// ---- FBs/FB_ECS_Keba_P30_noWrite.TcPOU
FUNCTION_BLOCK FB_ECS_Keba_P30_noWrite
VAR_INPUT PERSISTENT
	///{#lynus.ag#()} //Enable the Fuctionblock and his logic
	bEnable: BOOL;
	bEnable_write: BOOL;
	///With True its possible to invert all received power data from the electric meter
	bPowerDataInvers: BOOL;
	///Electric Fuse Line on wich the ECS is connected => 1 2 3 (If 0 then this charging station is not connected to a Electric Fuse Line)
	byElectricFuseLine: BYTE;
	///Failsafe Current when the connection between PLC and Charging station is interrupted. 0mA = CS Off, 6000mA - 32000mA
	uiFailsafeCurrent: UINT;
	///Failsafe Timeout when the connection between PLC and Charging station is interrupted. 10 - 600 sec
	uiFailsafeTimeOut: UINT := 10;
	///Number of EMS what control this Device.
	diNrOfEMS_IN: DINT;
	///Number of the electric meter for incoming power data. (Power Data for this Device)
	diNrOfEM_IN_CS: DINT;
	///IP Adress from the Keba charging station
	sIPAdress: STRING(15);
	///{#lynus.ag#()} //Setup charging station
	stSetupECS: ST_Setup_ECS;
END_VAR
VAR_OUTPUT
	///{#lynus.ag#()} //Electric charging station output data
	stDataECS: ST_ECS_Output;
	///Active Number from the Electric charging Function for using on other functions
	diNrOfECS_OUT: DINT;
	///Total Electric Power in kW read out directly from the Charging station. (Real time)
	lrTotalPowerECSRealTime: LREAL;
END_VAR
VAR
	///Function block for electric charging station

	fbCS: FB_ElectricChargingStation;
	///Function block to calcualte the number of the Device

	fbNumberDevice: FB_NumberOfDevice;
	///Digital Input from external loock signal
	fbDIExternalLock: FB_XL1XXX_DI;
	///Modbus Read Function (FC3)

	fbMBRead_FC3: FB_MBReadRegs;
	///Modbus Write Function (FC6)

	fbMBWrite_FC6: FB_MBWriteSingleReg;
	///Convert Word to Dword

	fbConvertWordToDword: FB_CV_WORD_TO_DWORD;
	///Timer for Delay between Requests

	timDelay: TON;
	///Timer for Timeout

	timTimeout: TON;
	///Timer to dissable the Function after Lynus_Standards.Constants_General.tTimeDissableLynusFunctions Days without connection to the Lynus Cloud

	timDissableFunctions: TON;
	///Timer to try reset the connection Flag on the GVL. (When somebody delete the Connection Function and make only a onlinechange)

	timResetConnectionOnGVL: TON;
	///Charging Time

	timChTimeSocket: TON;
	///Timer to start the state machine with Daley after enabling or after the system ist restartet

	timDelayStart: TON;
	///Timer to Close the Socket after to much Errors

	timCloseSocket: TON;
	///Internal positive Edge

	FPError_FC_3: R_TRIG;
	///Internal positive Edge

	FPError_FC_6: R_TRIG;
	///Internal positive Edge

	FPEnable: R_TRIG;
	///Function to save persistent data

	arrPD: ARRAY[1..16] OF FB_PersistentData_Number;
	///Function to save persistent string data

	fbPDString: FB_PersistentData_String;
	///Buffer with Data from FC3

	arrBuffer_FC3: ARRAY[1..2] OF WORD;
	///Error State from the charging station

	bErrorCS: BOOL;
	///Modbus TCP Function Error Counter																	

	byMBTCPErrorCounter: BYTE;
	///Wait in Step before start to clean data on PLC

	byWaitInStep: BYTE;
	///State machine to handle the data on the GVL

	iStateGVLData: INT;
	///State machine for read out Data over Modbus TCP

	iStateModbusRead: INT;
	///State machine for write Data over Modbus TCP

	iStateModbusWrite: INT;
	///State machine for error out Data over Modbus TCP	

	iStateModbusError: INT;
	///Variable to compare the state machine variable to set or reset the timeout timer

	iStateModbus_CP: INT;
	///Number of active batterys

	diNumberOfActiveBatterys: DINT;
	///Number of battery inverters that work in Emergency Power operation 

	diNumberOfBatteryInverterInEPO: DINT;
	///Loop to clean old data on GVL

	diLPForGVL: DINT;
	///Counter to clean old data on GVL

	diCounterForGVL: DINT;
	///Sum of the SOC from all batterys

	dwSumSOC: DWORD;
	///Charging State from the Keba Charger

	dwChargingState: DWORD;
	///Cable State from the Keba Charger

	dwCableState: DWORD;
	///Error Code from the Keba Charger

	dwErrorCode: DWORD;
	///Power from the ECS in W 

	rPowerECS: REAL;
	///Energy Counter Consumption in Wh

	lrTotalCounterEnergy_Consumption: LREAL;
	///Charged Energy from the active Session in Wh

	lrChargedEnergySession: LREAL;
	///Loop to check some data from batterys

	liLPBatteryData: LINT;
	///Loop to check if 1 or more battery inverters build a island grid

	liLPInEPO: LINT;
END_VAR
VAR PERSISTENT
	///Number of EMS what control this Device to compare with the original
	{attribute 'conditionalshow' := ''}
	diNrOfEMS_IN_CP: DINT;
END_VAR

//Creator : Stefan Lackner
//Company : EfficientIO
//Date : 14.05.2024
//Version : 1.0.0.1 based on V1.0.0.0

//With this Funcition its possible to communicate with a Keba P30 Charging station over Modbus TCP.
//Support the C-Series from Version 3.10.16 or higher
//Support the X-Series from Version 1.11 or higher
//Its possible to controll the charging station over the charge current
//When the Function send 0 Ampere is switched of, then the charging station is blocked and its not possible to charge
//The Communication is not so fast because in the Documentation they write that we can read every 500MS but we can write onle ever 5 seconds.
//We can read only 1 Register at each command. Its not possible to read more Registers with 1 command
//The Unit ID is always 255
//Also the Settings for Fail Save is includes in ths Fuction. The Failsave Current is set to uiFailsafeCurrent.
//Failsafe takes effect when the connection between the PLC and the charging station is interrupted. Timout is uiFailsafeTimeOut in seconds.

//Versions that are supported : 1.3

//NOTE for diNr.....Designation => 
//_IN = Here Data come in from other Functions or go out to other functions about the GVL
//_OUT = Here Data go out to other functions about the GVL

(*--------------------------------------------------------------------------------------------Limits-------------------------------------------------------------------------------------*)

diNrOfEMS_IN := LIMIT(0,diNrOfEMS_IN,Constants_Energy.diMaxNumberOfEMS);
diNrOfEM_IN_CS := LIMIT(0,diNrOfEM_IN_CS,Constants_Energy.diMaxNumberOfElectricMeters);
byElectricFuseLine := LIMIT(0,byElectricFuseLine,30);
IF uiFailsafeCurrent > 0 THEN 
	uiFailsafeCurrent := LIMIT(6000,uiFailsafeCurrent,32000);
END_IF 
uiFailsafeTimeOut := LIMIT(10,uiFailsafeTimeOut,600);	
		
(*------------------------------------------------------------------Power Data----------------------------------------------------------------------------*)

IF diNrOfEM_IN_CS <> 0 THEN
	//Energy Session Input data
	fbCS.bCalculateEnergySession := FALSE;
	fbCS.arrSocketPowerECS[1] := 0;
	fbCS.arrSocketPowerECS[2] := 0;
	fbCS.arrSocketPowerECS[3] := 0;
	fbCS.arrSocketPowerECS[4] := 0;
	fbCS.arrSocketEnergySession[1] := 0;
	fbCS.arrSocketEnergySession[2] := 0;
	fbCS.arrSocketEnergySession[3] := 0;
	fbCS.arrSocketEnergySession[4] := 0;
	IF NOT bPowerDataInvers THEN
		//Energy meter input data for cs Function block
		fbCS.lrCounterEnergyT1_Consumption := Lynus_Standards.GVL_Energy.stDataElectricMeters[diNrOfEM_IN_CS].lrCounterEnergyT1_Production * 1000;
		fbCS.lrCounterEnergyT2_Consumption := Lynus_Standards.GVL_Energy.stDataElectricMeters[diNrOfEM_IN_CS].lrCounterEnergyT2_Production * 1000;
		fbCS.lrCounterEnergyT1_Production := Lynus_Standards.GVL_Energy.stDataElectricMeters[diNrOfEM_IN_CS].lrCounterEnergyT1_Consumption * 1000;
		fbCS.lrCounterEnergyT2_Production := Lynus_Standards.GVL_Energy.stDataElectricMeters[diNrOfEM_IN_CS].lrCounterEnergyT1_Consumption * 1000;
		fbCS.lrTotalCounterEnergy_Consumption := Lynus_Standards.GVL_Energy.stDataElectricMeters[diNrOfEM_IN_CS].lrTotalCounterEnergy_Production * 1000;
		fbCS.lrTotalCounterEnergy_Production := Lynus_Standards.GVL_Energy.stDataElectricMeters[diNrOfEM_IN_CS].lrTotalCounterEnergy_Consumption * 1000;
		fbCS.lrTotalPowerECS := (Lynus_Standards.GVL_Energy.stDataElectricMeters[diNrOfEM_IN_CS].lrPower * 1000) * - 1;
	ELSE
		//Energy meter input data for cs Function block
		fbCS.lrCounterEnergyT1_Consumption := Lynus_Standards.GVL_Energy.stDataElectricMeters[diNrOfEM_IN_CS].lrCounterEnergyT1_Consumption * 1000;
		fbCS.lrCounterEnergyT2_Consumption := Lynus_Standards.GVL_Energy.stDataElectricMeters[diNrOfEM_IN_CS].lrCounterEnergyT2_Consumption * 1000;
		fbCS.lrCounterEnergyT1_Production := Lynus_Standards.GVL_Energy.stDataElectricMeters[diNrOfEM_IN_CS].lrCounterEnergyT1_Production * 1000;
		fbCS.lrCounterEnergyT2_Production := Lynus_Standards.GVL_Energy.stDataElectricMeters[diNrOfEM_IN_CS].lrCounterEnergyT2_Production * 1000;
		fbCS.lrTotalCounterEnergy_Consumption := Lynus_Standards.GVL_Energy.stDataElectricMeters[diNrOfEM_IN_CS].lrTotalCounterEnergy_Consumption * 1000;
		fbCS.lrTotalCounterEnergy_Production := Lynus_Standards.GVL_Energy.stDataElectricMeters[diNrOfEM_IN_CS].lrTotalCounterEnergy_Production * 1000;
		fbCS.lrTotalPowerECS := Lynus_Standards.GVL_Energy.stDataElectricMeters[diNrOfEM_IN_CS].lrPower * 1000;
	END_IF
ELSE
	//Energy meter input data for cs Function block
	fbCS.lrCounterEnergyT1_Consumption := lrTotalCounterEnergy_Consumption;
	fbCS.lrCounterEnergyT2_Consumption := 0;
	fbCS.lrCounterEnergyT1_Production := 0;
	fbCS.lrCounterEnergyT2_Production := 0;
	fbCS.lrTotalCounterEnergy_Consumption := lrTotalCounterEnergy_Consumption;
	fbCS.lrTotalCounterEnergy_Production := 0;
	fbCS.lrTotalPowerECS := rPowerECS;
	//Energy Session Input data
	fbCS.bCalculateEnergySession := FALSE;
	fbCS.arrSocketPowerECS[1] := rPowerECS;
	fbCS.arrSocketPowerECS[2] := 0;
	fbCS.arrSocketPowerECS[3] := 0;
	fbCS.arrSocketPowerECS[4] := 0;
	fbCS.arrSocketEnergySession[1] := lrChargedEnergySession;
	fbCS.arrSocketEnergySession[2] := 0;
	fbCS.arrSocketEnergySession[3] := 0;
	fbCS.arrSocketEnergySession[4] := 0;
END_IF			

(*-------------------------------------------------------------Calcualte the number of ECS---------------------------------------------------------------*)

fbNumberDevice(
	diActualNumberOfDevices:= Lynus_Standards.GVL_Energy.stNumberOfDevices.diNumberOfECS, 
	diMaxNumberOfDevices:= Constants_Energy.diMaxNumberOfElectricChargingStations, 
	udiCounterOnlineChange:= TwinCAT_SystemInfoVarList._AppInfo.OnlineChangeCnt, 
	bNumberIsCalculatet=> , 
	bFPNumberIsCalculatet=> , 
	bOnlineChange=> , 
	diNumberForThisDevice=> diNrOfECS_OUT, 
	diNumberOfTotalDevices=> );

//Write new Numer on GVL
IF fbNumberDevice.bFPNumberIsCalculatet THEN
	Lynus_Standards.GVL_Energy.stNumberOfDevices.diNumberOfECS := fbNumberDevice.diNumberOfTotalDevices;	
END_IF 

//Delete old Number on GVL
IF fbNumberDevice.bOnlineChange THEN 
	Lynus_Standards.GVL_Energy.stNumberOfDevices.diNumberOfECS := diNrOfECS_OUT;	
	iStateGVLData := 1;
END_IF

(*-------------------------------------------------------------Service from Backend is ready and check the connection to backen for dissabel/enable Function---------------------------------------------------------------*)

//Try to reset the variable for connection on the GVL. When all is normal then the Lynus Mqtt connection function set this variable to true in the next cycle
//When we have no connection to the backend then after Lynus_Standards.Constants_General.tTimeDissableLynusFunctions days the Function is dissabled with all of his functionalities
timResetConnectionOnGVL(IN:= NOT timResetConnectionOnGVL.Q, PT:= T#1H, Q=> , ET=> );
IF timResetConnectionOnGVL.Q THEN 
	Lynus_Standards.GVL_Communicator.bStateConnectionToEnableFunctions := FALSE; 
END_IF
IF NOT Lynus_Standards.GVL_Communicator.bStateConnectionToEnableFunctions THEN 
	timDissableFunctions.IN := TRUE; 
ELSE 
	timDissableFunctions.IN := FALSE; 
END_IF  
timDissableFunctions(	IN:= , 	
						PT:= Lynus_Standards.Constants_General.tTimeDissableLynusFunctions, 
						Q=> , 
						ET=> );
			
(*--------------------------------------------------------------------------------------------State Machine Read--------------------------------------------------------------------------------------*)

//Timer for Delay
timDelay(	IN:= , 
			PT:= T#750MS, 
			Q=> , 
			ET=> );

//Timer for Timeout in Statemachine
IF 	(iStateModbusRead > 0 AND iStateModbusRead <= 7 AND iStateModbusRead = iStateModbus_CP) OR
	(iStateModbusWrite > 0 AND iStateModbusWrite <= 2 AND iStateModbusWrite = iStateModbus_CP) THEN
		timTimeout.IN := TRUE;
ELSE	
		timTimeout.IN := FALSE;
END_IF
//Timeout Timer is dissabled when the Init Step is aktiv or the function is not enabled
IF (iStateModbusRead = 0 AND iStateModbusWrite = 0) OR NOT bEnable THEN 
	timTimeout.IN := FALSE; 
END_IF
timTimeout(	IN:= , 
			PT:= T#10S, 
			Q=> , 
			ET=> );

//Enable with Delay that not all sockets have to be created at the same time
timDelayStart(	IN:= bEnable, 
				PT:= T#20MS * diNrOfECS_OUT, 
				Q=> , 
				ET=> );
FPEnable(	CLK:= timDelayStart.Q, 
			Q=> );

IF FPEnable.Q AND iStateModbusRead = 0 AND iStateModbusWrite = 0 THEN 
	iStateModbusRead := 1; 
END_IF		
		
//Not Enabled
IF NOT bEnable THEN 
	iStateModbusRead := 0; 
	iStateModbusError := 0; 
	iStateModbusWrite := 0; 
END_IF		
		
CASE iStateModbusRead OF

	0://Init Step 
		iStateModbus_CP := 0;
		timDelay.IN := FALSE;
		fbMBRead_FC3.bExecute := FALSE;
		fbMBWrite_FC6.bExecute := FALSE;
		rPowerECS := 0;
		dwChargingState := 0;
		dwCableState := 0;	
		lrChargedEnergySession := 0;
	
	1://Charging State (Register 1000) !!!!Maybe 0 or 1....test it. Then change also the other Register Adresses!!!!!
		iStateModbus_CP := iStateModbusRead;

		//Start Read
		fbMBRead_FC3.nQuantity := 2;
		fbMBRead_FC3.nMBAddr := 1000;
		fbMBRead_FC3.bExecute := TRUE;
		fbMBRead_FC3.nUnitID := 255;
			
		IF fbMBRead_FC3.bBusy THEN 
			timDelay.IN := TRUE; 
		END_IF
		
		//Wait for Delay, copy Data and then next step
		IF NOT fbMBRead_FC3.bBusy AND NOT fbMBRead_FC3.bError AND timDelay.Q THEN
			//Charging State
			fbConvertWordToDword(wInputValue_1:= arrBuffer_FC3[1], wInputValue_2:= arrBuffer_FC3[2], eByteOrderForConvert:= eByteOrder.eBigEndian, dwOutputValue =>);
			dwChargingState := fbConvertWordToDword.dwOutputValue;
			
			//Go to Next Step
			fbMBRead_FC3.bExecute := FALSE;
			timDelay.IN := FALSE;		
			iStateModbusRead := 2;
		END_IF	

		//Error or Timeout
		IF FPError_FC_3.Q OR timTimeout.Q THEN
			iStateModbusError := 300;
		END_IF	
		
	2://Cable State (Register 1004)
		iStateModbus_CP := iStateModbusRead;

		//Start Read
		fbMBRead_FC3.nQuantity := 2;
		fbMBRead_FC3.nMBAddr := 1004;
		fbMBRead_FC3.bExecute := TRUE;
		fbMBRead_FC3.nUnitID := 255;
			
		IF fbMBRead_FC3.bBusy THEN 
			timDelay.IN := TRUE; 
		END_IF
		
		//Wait for Delay, copy Data and then next step
		IF NOT fbMBRead_FC3.bBusy AND NOT fbMBRead_FC3.bError AND timDelay.Q THEN
			//Cable State
			fbConvertWordToDword(wInputValue_1:= arrBuffer_FC3[1], wInputValue_2:= arrBuffer_FC3[2], eByteOrderForConvert:= eByteOrder.eBigEndian, dwOutputValue =>);
			dwCableState := fbConvertWordToDword.dwOutputValue;
			//Go to Next Step
			fbMBRead_FC3.bExecute := FALSE;
			timDelay.IN := FALSE;		
			iStateModbusRead := 3;
		END_IF	

		//Error or Timeout
		IF FPError_FC_3.Q OR timTimeout.Q THEN
			iStateModbusError := 300;
		END_IF	
		
	3://Error Code (Register 1006)
		iStateModbus_CP := iStateModbusRead;

		//Start Read
		fbMBRead_FC3.nQuantity := 2;
		fbMBRead_FC3.nMBAddr := 1006;
		fbMBRead_FC3.bExecute := TRUE;
		fbMBRead_FC3.nUnitID := 255;
			
		IF fbMBRead_FC3.bBusy THEN 
			timDelay.IN := TRUE; 
		END_IF
		
		//Wait for Delay, copy Data and then next step
		IF NOT fbMBRead_FC3.bBusy AND NOT fbMBRead_FC3.bError AND timDelay.Q THEN
			//Error Code
			fbConvertWordToDword(wInputValue_1:= arrBuffer_FC3[1], wInputValue_2:= arrBuffer_FC3[2], eByteOrderForConvert:= eByteOrder.eBigEndian, dwOutputValue =>);
			dwErrorCode := fbConvertWordToDword.dwOutputValue;
			//Go to Next Step
			fbMBRead_FC3.bExecute := FALSE;
			timDelay.IN := FALSE;		
			iStateModbusRead := 4;
		END_IF	

		//Error or Timeout
		IF FPError_FC_3.Q OR timTimeout.Q THEN
			iStateModbusError := 300;
		END_IF	
		
	4://Active Power (Register 1020)
		iStateModbus_CP := iStateModbusRead;

		//Start Read
		fbMBRead_FC3.nQuantity := 2;
		fbMBRead_FC3.nMBAddr := 1020;
		fbMBRead_FC3.bExecute := TRUE;
		fbMBRead_FC3.nUnitID := 255;
			
		IF fbMBRead_FC3.bBusy THEN 
			timDelay.IN := TRUE; 
		END_IF
		
		//Wait for Delay, copy Data and then next step
		IF NOT fbMBRead_FC3.bBusy AND NOT fbMBRead_FC3.bError AND timDelay.Q THEN
			//Active Power in mW
			fbConvertWordToDword(wInputValue_1:= arrBuffer_FC3[1], wInputValue_2:= arrBuffer_FC3[2], eByteOrderForConvert:= eByteOrder.eBigEndian, dwOutputValue =>);
			rPowerECS := DWORD_TO_REAL(fbConvertWordToDword.dwOutputValue);
			rPowerECS := rPowerECS / 1000;	
			//Go to Next Step
			fbMBRead_FC3.bExecute := FALSE;
			timDelay.IN := FALSE;		
			iStateModbusRead := 5;
		END_IF	

		//Error or Timeout
		IF FPError_FC_3.Q OR timTimeout.Q THEN
			iStateModbusError := 300;
		END_IF	
	
	5://Total Energy (Register 1036)
		iStateModbus_CP := iStateModbusRead;

		//Start Read
		fbMBRead_FC3.nQuantity := 2;
		fbMBRead_FC3.nMBAddr := 1036;
		fbMBRead_FC3.bExecute := TRUE;
		fbMBRead_FC3.nUnitID := 255;
			
		IF fbMBRead_FC3.bBusy THEN 
			timDelay.IN := TRUE; 
		END_IF
		
		//Wait for Delay, copy Data and then next step
		IF NOT fbMBRead_FC3.bBusy AND NOT fbMBRead_FC3.bError AND timDelay.Q THEN
			//Total Energy in Wh
			fbConvertWordToDword(wInputValue_1:= arrBuffer_FC3[1], wInputValue_2:= arrBuffer_FC3[2], eByteOrderForConvert:= eByteOrder.eBigEndian, dwOutputValue =>);
			lrTotalCounterEnergy_Consumption := DWORD_TO_LREAL(fbConvertWordToDword.dwOutputValue);
			//Go to Next Step
			fbMBRead_FC3.bExecute := FALSE;
			timDelay.IN := FALSE;		
			iStateModbusRead := 6;
		END_IF	

		//Error or Timeout
		IF FPError_FC_3.Q OR timTimeout.Q THEN
			iStateModbusError := 300;
		END_IF	
		
	6://Charged Energy from current charging session (Register 1502)
		iStateModbus_CP := iStateModbusRead;

		//Start Read
		fbMBRead_FC3.nQuantity := 2;
		fbMBRead_FC3.nMBAddr := 1502;
		fbMBRead_FC3.bExecute := TRUE;
		fbMBRead_FC3.nUnitID := 255;
			
		IF fbMBRead_FC3.bBusy THEN 
			timDelay.IN := TRUE; 
		END_IF
		
		//Wait for Delay, copy Data and then next step
		IF NOT fbMBRead_FC3.bBusy AND NOT fbMBRead_FC3.bError AND timDelay.Q THEN
			//Total Energy in Wh
			fbConvertWordToDword(wInputValue_1:= arrBuffer_FC3[1], wInputValue_2:= arrBuffer_FC3[2], eByteOrderForConvert:= eByteOrder.eBigEndian, dwOutputValue =>);
			lrChargedEnergySession := DWORD_TO_LREAL(fbConvertWordToDword.dwOutputValue);
			//Go to Next Step
			fbMBRead_FC3.bExecute := FALSE;
			timDelay.IN := FALSE;		
			iStateModbusRead := 7;
		END_IF	

		//Error or Timeout
		IF FPError_FC_3.Q OR timTimeout.Q THEN
			iStateModbusError := 300;
		END_IF	
		
	7://Wait 1 Step to reset the delay counter befor start to write
		iStateModbus_CP := iStateModbusRead;
		IF bEnable_write THEN 
			iStateModbusWrite := 1;
			//-1 because 0 is the Init Step for Read
			iStateModbusRead := - 1;
		ELSE
			iStateModbusRead := 1;
		END_IF				
		//Error on Master, changes on Inputs or Timeout
		IF timTimeout.Q THEN 
			iStateModbusError := 300;	 
		END_IF

END_CASE

(*------------------------------------------------------------------Error and Warning----------------------------------------------------------------------------*)	
 
IF dwChargingState = 4 OR dwErrorCode <> 0 THEN 
	bErrorCS := TRUE; 
ELSE 
	bErrorCS := FALSE; 
END_IF

IF timDissableFunctions.Q THEN 
	fbCS.bWarning := TRUE; 
	fbCS.iWarningCode := 0; 
ELSE 
	fbCS.bWarning := FALSE; 
END_IF   
IF Lynus_Standards.GVL_Energy.stNumberOfDevices.diNumberOfECS > Constants_Energy.diMaxNumberOfElectricChargingStations OR bErrorCS OR byMBTCPErrorCounter > 10 THEN 
	fbCS.bError := TRUE;
ELSE 
	fbCS.bError := FALSE;
	fbCS.iErrorCode := 0;
END_IF

IF Lynus_Standards.GVL_Energy.stNumberOfDevices.diNumberOfECS > Constants_Energy.diMaxNumberOfElectricChargingStations THEN 
	fbCS.iErrorCode := 1;
ELSIF bErrorCS OR byMBTCPErrorCounter > 10 THEN 
	fbCS.iErrorCode := 0; 
END_IF

(*------------------------------------------------------------------Logic----------------------------------------------------------------------------*)

//Calcualte the total SOC if we have more then 1 battery in our system
diNumberOfActiveBatterys := 0;
dwSumSOC := 0;
FOR liLPBatteryData := 1 TO Constants_Energy.diMaxNumberOfBatterys BY 1 DO
	IF Lynus_Standards.GVL_Energy.stDataOfBatterys[diNrOfEMS_IN,liLPBatteryData].bEnabled THEN 
		diNumberOfActiveBatterys := diNumberOfActiveBatterys + 1; 
	END_IF
	dwSumSOC := dwSumSOC + Lynus_Standards.GVL_Energy.stDataOfBatterys[diNrOfEMS_IN,liLPBatteryData].dwSOC;
END_FOR
	
IF diNumberOfActiveBatterys > 0 THEN
	fbCS.dwBatterySOC := DINT_TO_DWORD(DWORD_TO_DINT(dwSumSOC) / diNumberOfActiveBatterys);
ELSE
	fbCS.dwBatterySOC := 100;	//When we have no battery in the ems system
END_IF

//Check if one or more Batterysystems or batteryinverter make island mode
diNumberOfBatteryInverterInEPO := 0;
FOR liLPInEPO := 1 TO Constants_Energy.diMaxNumberOfBatteryInverters BY 1 DO
	IF Lynus_Standards.GVL_Energy.stDataOfBatteryInverters[diNrOfEMS_IN,liLPInEPO].bWorkOnIslandMode THEN 
		fbCS.bEPOIsActive := TRUE; diNumberOfBatteryInverterInEPO := diNumberOfBatteryInverterInEPO + 1; 
	END_IF
END_FOR 
IF diNumberOfBatteryInverterInEPO <= 0 THEN 
	fbCS.bEPOIsActive := FALSE; 
END_IF

//Digital input for external lock signal
fbDIExternalLock(bInvers:= FALSE, bSignal=> );

//Car connected to the ECS
IF dwCableState = 5 OR dwCableState = 7 THEN 
	fbCS.bCarConnected := TRUE; 
ELSE 
	fbCS.bCarConnected := FALSE; 
END_IF

//Charging time
IF dwChargingState = 3 OR dwCableState = 7 THEN 
	timChTimeSocket.IN := TRUE; 
ELSE 
	timChTimeSocket.IN := FALSE; 
END_IF

IF timChTimeSocket.IN THEN 
	fbCS.arrSocketChargingTimeInput[1] := TIME_TO_REAL(timChTimeSocket.ET) / 60000; 
END_IF
fbCS.arrSocketChargingTimeInput[2] := 0;
fbCS.arrSocketChargingTimeInput[3] := 0;
fbCS.arrSocketChargingTimeInput[4] := 0;

timChTimeSocket(	IN:= , 
					PT:= T#24H, 
					Q=> , 
					ET=> );

//Mode 3 State
//Default set to No Informantion
fbCS.arrSocketMode3StateECS[1] := '';
//Ready or Free
IF dwChargingState = 2 THEN 
	fbCS.arrSocketMode3StateECS[1] := 'A'; 
END_IF
//Car Connected
IF dwCableState = 5 OR dwCableState = 7 THEN 
	fbCS.arrSocketMode3StateECS[1] := 'B1'; 
END_IF
//Charging
IF dwChargingState = 3 OR dwCableState = 7 THEN 
	fbCS.arrSocketMode3StateECS[1] := 'C2'; 
END_IF
//Error
IF dwChargingState = 4 OR dwErrorCode <> 0 THEN 
	fbCS.arrSocketMode3StateECS[1] := 'F'; 
END_IF 

fbCS.arrSocketMode3StateECS[2] := '';
fbCS.arrSocketMode3StateECS[3] := '';
fbCS.arrSocketMode3StateECS[4] := '';

//SOC Car
fbCS.arrSOCCar[1] := 0;
fbCS.arrSOCCar[2] := 0;
fbCS.arrSOCCar[3] := 0;
fbCS.arrSOCCar[4] := 0;

//Functionblock ECS
fbCS(
	bEnable:= bEnable AND NOT timDissableFunctions.Q, 
	bError:= ,
	bWarning := ,
	bEPOIsActive:= , 
	bExternalLock:= fbDIExternalLock.bSignal, 
	bCarConnected:= , 
	bWriteWithDelay:= TRUE, 
	bCalculateEnergySession:= ,
	iErrorCode:= , 
	iWarningCode:= , 
	arrSocketChargingTimeInput:= ,
	arrSOCCar:= , 
	dwBatterySOC:= , 
	lrTotalCounterEnergy_Consumption:= , 
	lrTotalCounterEnergy_Production:= , 
	lrCounterEnergyT1_Consumption:= , 
	lrCounterEnergyT2_Consumption:= , 
	lrCounterEnergyT1_Production:= , 
	lrCounterEnergyT2_Production:= , 
	lrTotalPowerECS:= , 
	arrSocketEnergySession:= ,
	rTargetPower:= Lynus_Standards.GVL_Energy.stDataElectricChargingStations[diNrOfEMS_IN,diNrOfECS_OUT].rTargetPowerEMS, 
	rSupplyVoltage:= 692, 
	rMinCurrent:= 6, 
	tTimDelayOutput:= T#5S, 
	tDelayError:= T#5S,
	arrSocketMode3StateECS:= ,
	arrSocketPowerECS:= ,
	stSetupECS:= stSetupECS, 
	stDataECSOut=> , 
	stDataECSOutDelay=> stDataECS);

//Real time Power for Output
lrTotalPowerECSRealTime := fbCS.stDataECSOut.lrTotalPower;
	
(*------------------------------------------------------------------------------------------State Machine Write---------------------------------------------------------------------------------------------*)	

CASE iStateModbusWrite OF	

	1://Set the charging current (Reg 5004)
		iStateModbus_CP := iStateModbusWrite;
		
		fbMBWrite_FC6.nMBAddr := 5004;
		fbMBWrite_FC6.bExecute := TRUE;
		fbMBWrite_FC6.nUnitID := 255;
		//Charge Current in mA
		fbMBWrite_FC6.nValue := REAL_TO_WORD(fbCS.stDataECSOut.rTargetChargeCurrent * 1000);
		
		IF fbMBWrite_FC6.bBusy THEN 
			timDelay.IN := TRUE; 
		END_IF

		//Wait for Delay and then next step
		IF NOT fbMBWrite_FC6.bBusy AND NOT fbMBWrite_FC6.bError AND timDelay.Q THEN
			fbMBWrite_FC6.bExecute := FALSE;
			timDelay.IN := FALSE;
			//Go to Next Step
			iStateModbusWrite := 2;
		END_IF
				
		//Error or Timout
		IF FPError_FC_6.Q OR timTimeout.Q THEN
			iStateModbusError := 300;
		END_IF
	
	2://Enable/Dissable Charging station (Reg 5014)
		iStateModbus_CP := iStateModbusWrite;
		
		fbMBWrite_FC6.nMBAddr := 5014;
		fbMBWrite_FC6.bExecute := TRUE;
		fbMBWrite_FC6.nUnitID := 255;
		//Enable and Dissable the Charging station
		IF fbCS.stDataECSOut.rTargetChargeCurrent <> 0 THEN 
			//Enable
			fbMBWrite_FC6.nValue := 1;
		ELSE
			//Dissable
			fbMBWrite_FC6.nValue := 0;
		END_IF
		
		IF fbMBWrite_FC6.bBusy THEN 
			timDelay.IN := TRUE; 
		END_IF

		//Wait for Delay and then next step
		IF NOT fbMBWrite_FC6.bBusy AND NOT fbMBWrite_FC6.bError AND timDelay.Q THEN
			fbMBWrite_FC6.bExecute := FALSE;
			timDelay.IN := FALSE;
			//Go to Next Step
			iStateModbusWrite := 3;
		END_IF
				
		//Error or Timout
		IF FPError_FC_6.Q OR timTimeout.Q THEN
			iStateModbusError := 300;
		END_IF
		
	3://Failsafe current (Reg 5016)
		iStateModbus_CP := iStateModbusWrite;
		
		fbMBWrite_FC6.nMBAddr := 5016;
		fbMBWrite_FC6.bExecute := TRUE;
		fbMBWrite_FC6.nUnitID := 255;
		//Failsafe current in mA
		fbMBWrite_FC6.nValue := uiFailsafeCurrent;
	
		IF fbMBWrite_FC6.bBusy THEN 
			timDelay.IN := TRUE; 
		END_IF

		//Wait for Delay and then next step
		IF NOT fbMBWrite_FC6.bBusy AND NOT fbMBWrite_FC6.bError AND timDelay.Q THEN
			fbMBWrite_FC6.bExecute := FALSE;
			timDelay.IN := FALSE;
			//Go to Next Step
			iStateModbusWrite := 3;
		END_IF
				
		//Error or Timout
		IF FPError_FC_6.Q OR timTimeout.Q THEN
			iStateModbusError := 300;
		END_IF	
		
	4://Failsafe Timeout (Reg 5018)
		iStateModbus_CP := iStateModbusWrite;
		
		fbMBWrite_FC6.nMBAddr := 5018;
		fbMBWrite_FC6.bExecute := TRUE;
		fbMBWrite_FC6.nUnitID := 255;
		//Failsafe Timeout in sec.
		fbMBWrite_FC6.nValue := uiFailsafeTimeOut;
	
		IF fbMBWrite_FC6.bBusy THEN 
			timDelay.IN := TRUE; 
		END_IF

		//Wait for Delay and then next step
		IF NOT fbMBWrite_FC6.bBusy AND NOT fbMBWrite_FC6.bError AND timDelay.Q THEN
			fbMBWrite_FC6.bExecute := FALSE;
			timDelay.IN := FALSE;
			byMBTCPErrorCounter := 0; 
			//Restart from new with the Read out part
			iStateModbusRead := 1;
			iStateModbusWrite := 0;
		END_IF
				
		//Error or Timout
		IF FPError_FC_6.Q OR timTimeout.Q THEN
			iStateModbusError := 300;
		END_IF	
		
END_CASE	
	
(*------------------------------------------------------------------------------------------State Machine Error---------------------------------------------------------------------------------------------*)	

CASE iStateModbusError OF
	
	300://Error
		iStateModbus_CP := iStateModbusError;
		timDelay.IN := FALSE;
		fbMBRead_FC3.bExecute := FALSE;
		fbMBWrite_FC6.bExecute := FALSE;
		byMBTCPErrorCounter := byMBTCPErrorCounter + 1;
		byMBTCPErrorCounter := LIMIT(0,byMBTCPErrorCounter,11); 		
		//Restart from new with the Read out part after an Error
		IF byMBTCPErrorCounter < 10 THEN
			iStateModbusRead := 1;	
			iStateModbusError := 0;
			iStateModbusWrite := 0;
		ELSE
			//Wait here in the Error State for the Delay Timer and then we dont have a Timeout Error
			iStateModbusRead := - 1;
			iStateModbusWrite := - 1;
			//Start from New when the Delay is paste
			IF timCloseSocket.Q THEN
				iStateModbusRead := 1;	
				iStateModbusError := 0;
				iStateModbusWrite := 0;	
				byMBTCPErrorCounter := 0;
			END_IF
		END_IF
		
END_CASE

//Timer to close the Socket after to much TCP Errors and reopen a new one
timCloseSocket(	IN:= byMBTCPErrorCounter > 10 AND fbCS.stDataECSOut.bEnabled, 
				PT:= T#1M, 
				Q=> , 
				ET=> );

(*------------------------------------------------------------------------------------------Modbus TCP Functions---------------------------------------------------------------------------------------------*)

fbMBRead_FC3(	sIPAddr:= sIPAdress, 
				nTCPPort:= 502,
				cbLength:= SIZEOF(arrBuffer_FC3), 
				pDestAddr:= ADR(arrBuffer_FC3), 
				tTimeout:= T#5S );
FPError_FC_3(	CLK:= fbMBRead_FC3.bError, 
				Q=> );		

fbMBWrite_FC6(	sIPAddr:= sIPAdress, 
				nTCPPort:= 502, 
				tTimeout:= T#5S);	
FPError_FC_6(	CLK:= fbMBWrite_FC6.bError, 
				Q=> );

(*-----------------------------------------------------------Handle data to Global structure for electric charging stations-----------------------------------------------------------------*)

//Delte al old Data on GVL after a online change or change on the variable diNrOfEMS_IDOD
IF diNrOfEMS_IN <> diNrOfEMS_IN_CP AND iStateGVLData = 0 THEN 
	iStateGVLData := 10; 
END_IF 

CASE iStateGVLData OF
	
	0://Init Step
		byWaitInStep := 0;
		diCounterForGVL := 1;
	
	1://Wait for 4 Steps before clean al Data on GVL
		byWaitInStep := byWaitInStep + 1;
		IF byWaitInStep >= 4 AND fbNumberDevice.bNumberIsCalculatet THEN 
			iStateGVLData := 2; 
		END_IF
		//To much Devices, back to the Init step
		IF byWaitInStep >= 4 AND NOT fbNumberDevice.bNumberIsCalculatet THEN 
			iStateGVLData := 0; 
		END_IF	
			
	2://Clear all Data in GVL
		FOR diLPForGVL := 1 TO Constants_Energy.diMaxNumberOfEMS BY 1 DO 
			Lynus_Standards.GVL_Energy.stDataElectricChargingStations[diLPForGVL,diCounterForGVL].bEnabled := FALSE;
			Lynus_Standards.GVL_Energy.stDataElectricChargingStations[diLPForGVL,diCounterForGVL].bIsControllable := FALSE;
			Lynus_Standards.GVL_Energy.stDataElectricChargingStations[diLPForGVL,diCounterForGVL].byErrorWarning := 0;
			Lynus_Standards.GVL_Energy.stDataElectricChargingStations[diLPForGVL,diCounterForGVL].byPriority := 0;
			Lynus_Standards.GVL_Energy.stDataElectricChargingStations[diLPForGVL,diCounterForGVL].lrPower := 0;
			Lynus_Standards.GVL_Energy.stDataElectricChargingStations[diLPForGVL,diCounterForGVL].lrPowerConsumption := 0;
			Lynus_Standards.GVL_Energy.stDataElectricChargingStations[diLPForGVL,diCounterForGVL].lrPowerProduction := 0;
			Lynus_Standards.GVL_Energy.stDataElectricChargingStations[diLPForGVL,diCounterForGVL].rMaxPower := 0;
			Lynus_Standards.GVL_Energy.stDataElectricChargingStations[diLPForGVL,diCounterForGVL].byElectricFuseLine := 0;
			//Set also the target value from ems back here to 0 and not in EMS function because EMS is in Standy when we have a online change (Problem when we delete a ems function and make a online change)
			Lynus_Standards.GVL_Energy.stDataElectricChargingStations[diLPForGVL,diCounterForGVL].rTargetPowerEMS := 0;	
		END_FOR
		
		//Counter for ECS
		diCounterForGVL := diCounterForGVL + 1;
		diCounterForGVL := LIMIT(0,diCounterForGVL,Constants_Energy.diMaxNumberOfElectricChargingStations);
		//Back to the init step
		IF diCounterForGVL >= Constants_Energy.diMaxNumberOfElectricChargingStations THEN 
			iStateGVLData := 0; 
		END_IF

	10://Clear old Data on GVL 		
		Lynus_Standards.GVL_Energy.stDataElectricChargingStations[diNrOfEMS_IN_CP,diNrOfECS_OUT].bEnabled := FALSE;
		Lynus_Standards.GVL_Energy.stDataElectricChargingStations[diNrOfEMS_IN_CP,diNrOfECS_OUT].bIsControllable := FALSE;
		Lynus_Standards.GVL_Energy.stDataElectricChargingStations[diNrOfEMS_IN_CP,diNrOfECS_OUT].byErrorWarning := 0;
		Lynus_Standards.GVL_Energy.stDataElectricChargingStations[diNrOfEMS_IN_CP,diNrOfECS_OUT].byPriority := 0;
		Lynus_Standards.GVL_Energy.stDataElectricChargingStations[diNrOfEMS_IN_CP,diNrOfECS_OUT].lrPower := 0;
		Lynus_Standards.GVL_Energy.stDataElectricChargingStations[diNrOfEMS_IN_CP,diNrOfECS_OUT].lrPowerConsumption := 0;
		Lynus_Standards.GVL_Energy.stDataElectricChargingStations[diNrOfEMS_IN_CP,diNrOfECS_OUT].lrPowerProduction := 0;
		Lynus_Standards.GVL_Energy.stDataElectricChargingStations[diNrOfEMS_IN_CP,diNrOfECS_OUT].rMaxPower := 0;
		Lynus_Standards.GVL_Energy.stDataElectricChargingStations[diNrOfEMS_IN_CP,diNrOfECS_OUT].byElectricFuseLine := 0;
		
		diNrOfEMS_IN_CP := diNrOfEMS_IN;
		//Back to the init step
		iStateGVLData := 0;

END_CASE 	 

IF diNrOfECS_OUT > 0 AND fbNumberDevice.bNumberIsCalculatet AND diNrOfEMS_IN > 0 THEN
	Lynus_Standards.GVL_Energy.stDataElectricChargingStations[diNrOfEMS_IN,diNrOfECS_OUT].bEnabled := fbCS.stDataECSOut.bEnabled;
	Lynus_Standards.GVL_Energy.stDataElectricChargingStations[diNrOfEMS_IN,diNrOfECS_OUT].bIsControllable := TRUE;
	Lynus_Standards.GVL_Energy.stDataElectricChargingStations[diNrOfEMS_IN,diNrOfECS_OUT].byErrorWarning := fbCS.stDataECSOut.byErrorWarning;
	Lynus_Standards.GVL_Energy.stDataElectricChargingStations[diNrOfEMS_IN,diNrOfECS_OUT].byPriority := fbCS.stDataECSOut.byPriority;
	Lynus_Standards.GVL_Energy.stDataElectricChargingStations[diNrOfEMS_IN,diNrOfECS_OUT].lrPower := fbCS.stDataECSOut.lrTotalPower;
	Lynus_Standards.GVL_Energy.stDataElectricChargingStations[diNrOfEMS_IN,diNrOfECS_OUT].lrPowerConsumption := fbCS.stDataECSOut.lrTotalPowerConsumption;
	Lynus_Standards.GVL_Energy.stDataElectricChargingStations[diNrOfEMS_IN,diNrOfECS_OUT].lrPowerProduction := fbCS.stDataECSOut.lrTotalPowerProduction;
	Lynus_Standards.GVL_Energy.stDataElectricChargingStations[diNrOfEMS_IN,diNrOfECS_OUT].rMaxPower := fbCS.stDataECSOut.rMaxPower;	
	Lynus_Standards.GVL_Energy.stDataElectricChargingStations[diNrOfEMS_IN,diNrOfECS_OUT].byElectricFuseLine := byElectricFuseLine;
END_IF 

(*----------------------------------------------------------Save persistent data----------------------------------------------------------------*)

arrPD[1](lrValue:= BOOL_TO_LREAL(bEnable), bEventBasedActive=> );
arrPD[2](lrValue:= BOOL_TO_LREAL(bPowerDataInvers), bEventBasedActive=> );
arrPD[3](lrValue:= DINT_TO_LREAL(diNrOfEMS_IN), bEventBasedActive=> );
arrPD[4](lrValue:= DINT_TO_LREAL(diNrOfEM_IN_CS), bEventBasedActive=> );
arrPD[5](lrValue:= BOOL_TO_LREAL(stSetupECS.bManualyOn), bEventBasedActive=> );
arrPD[6](lrValue:= BOOL_TO_LREAL(stSetupECS.bOnEmergPowerOff), bEventBasedActive=> );
arrPD[7](lrValue:= BYTE_TO_LREAL(stSetupECS.byCSMinPower), bEventBasedActive=> );
arrPD[8](lrValue:= BYTE_TO_LREAL(stSetupECS.byDisableSOC), bEventBasedActive=> );
arrPD[9](lrValue:= BYTE_TO_LREAL(stSetupECS.byEnableSOC), bEventBasedActive=> );
arrPD[10](lrValue:= BYTE_TO_LREAL(stSetupECS.byManualyTargetPower), bEventBasedActive=> );
arrPD[11](lrValue:= BYTE_TO_LREAL(stSetupECS.byPriority), bEventBasedActive=> );
arrPD[12](lrValue:= REAL_TO_LREAL(stSetupECS.rMaxPower), bEventBasedActive=> );
arrPD[13](lrValue:= DINT_TO_LREAL(diNrOfEMS_IN_CP), bEventBasedActive=> );
arrPD[14](lrValue:= BYTE_TO_LREAL(byElectricFuseLine), bEventBasedActive=> );
arrPD[15](lrValue:= UINT_TO_LREAL(uiFailsafeCurrent), bEventBasedActive=> );
arrPD[16](lrValue:= UINT_TO_LREAL(uiFailsafeTimeOut), bEventBasedActive=> );
fbPDString(sText:= sIPAdress, bEventBasedActive=> );

END_FUNCTION_BLOCK

// ---- POUs/prgComEffIO.TcPOU
PROGRAM prgComEffIO
VAR
	fbCom		: FB_MqttCommunicator_V2;
	
END_VAR


fbCom(
	bConnect:= TRUE, 
	strAuthKey:= 'EIO08031879806', 
	sUserName:= 'c0c17b06-0bdb-4698-a461-74f056a13e0b', 
	sUserPassword:= '80a8f7a1-49f9-455c-8c7e-584508cad010', 
	eSavePositionCertificate:= eSavePositionOnPLC.ePostionC,  
	time_HeartBeat_sec:= T#15S, 
	bConnected=> , 
	bError=> , 
	hrErrorCode=> , 
	eConnectionState=> , 
	eErrorMessage_Out=> );

END_PROGRAM

// ---- FBs/FB_Symo_PV_Inverter_FLOAT_1_DM_30_Inverter_1.TcPOU
{attribute 'hide_all_locals'}
FUNCTION_BLOCK FB_Symo_PV_Inverter_FLOAT_1_DM_30_Inverter_1
VAR_INPUT PERSISTENT
	bEnable						: BOOL;												//True = Function is enabled, FALSE = Function is dissabled, no new Data
	sIPAdress					: STRING(15);										//IP Adress from the Inverter
	arrUnitID_Inverter			: ARRAY[1..30] OF BYTE;								//Array with the Unit ID's from each Inverter (Max 30 Inverters) (ID = 1 to 247) (0 = No Inverter)
END_VAR
VAR_OUTPUT
	arrDataSymo10				: ARRAY[1..30] OF ST_Symo_PV_OutData;				//Output structure with Data from Symo 10
	stDataEMPower_PV			: ST_ElectricMeter_Output_Power;					//Output structure with Data from Electric Meter PV (Power Data)
	stDataEMCounter_PV			: ST_ElectricMeter_Output_Counter;					//Output structure with Data from Electric Meter PV (Counter Data)
	diNrOfEM_OUT_PV				: DINT;												//Active Number from the Electric Meter for using on other functions
END_VAR
VAR
	fbElMeter					: FB_ElectricMeter;									//Electric Meter Function 
	fbNumberDevice				: FB_NumberOfDevice;								//Function block to calcualte the number of the Device
	fbConvertEnergyRegister		: FB_CV_WORD_TO_DWORD;								//Convert function
	fbMBRead_FC3				: FB_MBReadRegs;									//Modbus Read Function (FC3)
	timDelay					: TON;												//Timer for Delay between Requests
	timTimeout					: TON;												//Timer for Timeout
	timDissableFunctions		: TON;												//Timer to dissable the Function after Lynus_Standards.Constants_General.tTimeDissableLynusFunctions Days without connection to the Lynus Cloud
	timResetConnectionOnGVL		: TON;												//Timer to try reset the connection Flag on the GVL. (When somebody delete the Connection Function and make only a onlinechange)
	FPEnable					: R_TRIG;											//Internal positive Edge
	FPError_FC_3				: R_TRIG;											//Internal positive Edge
	PD_String					: FB_PersistentData_String;							//Function to save persistent data 
	stFloat						: ST_UN_FLOAT_CONVERT_DWORD_REAL;					//Convert the Float Raw Value
	arrBuffer_FC3				: ARRAY[1..47] OF WORD;								//Buffer with Data from FC3
	arrUnitID_Inverter_CP		: ARRAY[1..30] OF BYTE;								//Array with unit IDs to compare it when we have a change on the Inputs
	arrCurrentL1				: ARRAY[1..30] OF LREAL;							//Array with the Current from L1 from each Inverter
	arrCurrentL2				: ARRAY[1..30] OF LREAL;							//Array with the Current from L2 from each Inverter
	arrCurrentL3				: ARRAY[1..30] OF LREAL;							//Array with the Current from L3 from each Inverter
	arrVoltageL1L2				: ARRAY[1..30] OF LREAL;							//Array with the Voltage from L1-L2 from each Inverter
	arrVoltageL2L3				: ARRAY[1..30] OF LREAL;							//Array with the Voltage from L2-L3 from each Inverter
	arrVoltageL3L1				: ARRAY[1..30] OF LREAL;							//Array with the Voltage from L3-L1 from each Inverter
	arrVoltageL1N				: ARRAY[1..30] OF LREAL;							//Array with the Voltage from L1-N from each Inverter
	arrVoltageL2N				: ARRAY[1..30] OF LREAL;							//Array with the Voltage from L2-N from each Inverter
	arrVoltageL3N				: ARRAY[1..30] OF LREAL;							//Array with the Voltage from L3-N from each Inverter
	arrACPower					: ARRAY[1..30] OF LREAL;							//Array with the AC Power from each Inverter
	arrFrequency				: ARRAY[1..30] OF LREAL;							//Array with the Frequency from each Inverter
	arrApparentPower			: ARRAY[1..30] OF LREAL;							//Array with the Apparent Power from each Inverter
	arrReactivePower			: ARRAY[1..30] OF LREAL;							//Array with the Reactive Power from each Inverter
	arrProductionEnergy			: ARRAY[1..30] OF LREAL;							//Array with the Production Energy from each Inverter
	arrPD						: ARRAY[1..31] OF FB_PersistentData_Number;			//Function to save persistent data
	bErrorDevice				: BOOL;												//When 1 or more Inverters has a Error, then thsi Flag is true
	byInverterInProgress		: BYTE;												//Shows what Inverter is at the moment in Progress in the State machine to read out the data
	byTotalInverter				: BYTE;												//Summ of total Inverters. (Depends on the unit IDs that are not 0.) 
	byLPForInverter				: BYTE; 											//Variable for Loop to calculate some things for the Inverters
	byWaitInStep				: BYTE;												//Wait in Step before start to clean data on PLC
	iStateGVLData				: INT;												//State machine to handle the data on the GVL
	iStateModbus				: INT;												//State variable for Statemachine
	iStateModbus_CP				: INT;												//Compare State variable
	diCounterForGVL				: DINT;												//Counter to clean old data on GVL
	lrCheckValue				: LREAL;											//Internal Value to check the value before convert
	lrCounterEnergyProduction	: LREAL;											//Check counter state before write new one
END_VAR

//Creator : Kai Ebensperger
//Company : Lynus AG
//Date : 28.04.2021
//Version : 1.0.0.0

//With this function its possible to read out values from the Symo 10 PV Inverter from the factory Fronius
//This Function read out the Values from 1 Fronius Datamanager with maximal 30 Inverter.
//The protocol to the Inverter is Modbus TCP
//Versions that are supported : 1.1.5-0
//Attention. To access the registers, an offset of 1 must always be subtracted. Register 40001 would then be on register 40000.
//This Function use the FLOAT Format
//You can query the register data of the individual devices using the Modbus device ID (UnitID).
//Each inverter has its own number stored on the display under "Setup" -> "Datcom"-> "Inverter number".
//Inverter number 00 = Modbus ID 100
//Inverter number 01 = Modbus ID 01
//Inverter number 02 = Modbus ID 02 etc.
//Internal in the GVL this function is 1 PV Plant. We display the summ ov all values from each Inverter

//Changes about AC power
//Date : 29.03.2020
//Version : 1.1.0.0

//NOTE for diNr.....Designation => 
//_IN = Here Data come in from other Functions or go out to other functions about the GVL
//_OUT = Here Data go out to other functions about the GVL

(*------------------------------------------------------------------------------------------General Input Part---------------------------------------------------------------------------------------------*)

//Check limitation
FOR byLPForInverter := 1 TO 30 BY 1 DO
	arrUnitID_Inverter[byLPForInverter] := LIMIT(0,arrUnitID_Inverter[byLPForInverter],247);
END_FOR

(*-------------------------------------------------------------Calcualte the number of EM System---------------------------------------------------------------*)

fbNumberDevice(
	diActualNumberOfDevices:= Lynus_Standards.GVL_Energy.stNumberOfDevices.diNumberOfElectricMeters, 
	diMaxNumberOfDevices:= Constants_Energy.diMaxNumberOfElectricMeters, 
	udiCounterOnlineChange:= TwinCAT_SystemInfoVarList._AppInfo.OnlineChangeCnt, 
	bNumberIsCalculatet=> , 
	bFPNumberIsCalculatet=> , 
	bOnlineChange=> , 
	diNumberForThisDevice=> diNrOfEM_OUT_PV, 
	diNumberOfTotalDevices=> );

//Write new Numer on GVL
IF fbNumberDevice.bFPNumberIsCalculatet THEN
	Lynus_Standards.GVL_Energy.stNumberOfDevices.diNumberOfElectricMeters := fbNumberDevice.diNumberOfTotalDevices;	
END_IF 

//Delete old Number on GVL
IF fbNumberDevice.bOnlineChange THEN 
	Lynus_Standards.GVL_Energy.stNumberOfDevices.diNumberOfElectricMeters := diNrOfEM_OUT_PV;	
		iStateGVLData := 1; 
END_IF

(*-------------------------------------------------------------Service from Backend is ready and check the connection to backen for dissabel/enable Function---------------------------------------------------------------*)

//Try to reset the variable for connection on the GVL. When all is normal then the Lynus Mqtt connection function set this variable to true in the next cycle
//When we have no connection to the backend then after Lynus_Standards.Constants_General.tTimeDissableLynusFunctions days the Function is dissabled with all of his functionalities
timResetConnectionOnGVL(IN:= NOT timResetConnectionOnGVL.Q, PT:= T#1H, Q=> , ET=> );
	IF timResetConnectionOnGVL.Q THEN Lynus_Standards.GVL_Communicator.bStateConnectionToEnableFunctions := FALSE; END_IF
		IF NOT Lynus_Standards.GVL_Communicator.bStateConnectionToEnableFunctions THEN timDissableFunctions.IN := TRUE; ELSE timDissableFunctions.IN := FALSE; END_IF  
			timDissableFunctions(IN:= , PT:= Lynus_Standards.Constants_General.tTimeDissableLynusFunctions, Q=> , ET=> );

(*------------------------------------------------------------------------------------------Calcualte the Max Number of Inverters---------------------------------------------------------------------------------------------*)
	
byTotalInverter := 0;
	FOR byLPForInverter := 1 TO 30 BY 1 DO
		IF arrUnitID_Inverter[byLPForInverter] <> 0 THEN byTotalInverter := byTotalInverter + 1; END_IF 
	END_FOR	
	
(*------------------------------------------------------------------------------------------State Machine---------------------------------------------------------------------------------------------*)
	
//Enable
FPEnable(CLK:= bEnable, Q=> );
	IF FPEnable.Q AND iStateModbus = 0 AND byTotalInverter > 0 THEN iStateModbus := 1; END_IF
		IF NOT bEnable OR timDissableFunctions.Q OR byTotalInverter = 0 OR MEMCMP(ADR(arrUnitID_Inverter),ADR(arrUnitID_Inverter_CP),SIZEOF(arrUnitID_Inverter_CP)) <> 0 THEN iStateModbus := 0; END_IF

//Timer for delay
timDelay(IN:= , PT:= T#50MS, Q=> , ET=> );	

//Timer for Timeout in Statemachine
	IF iStateModbus = iStateModbus_CP THEN timTimeout.IN := TRUE; ELSE timTimeout.IN := FALSE; END_IF
		IF iStateModbus = 0 THEN timTimeout.IN := FALSE; END_IF
timTimeout(IN:= , PT:= T#20S, Q=> , ET=> );	

//Statemachine
CASE iStateModbus OF
	
	0://Init Step
		iStateModbus_CP := iStateModbus;
			timDelay.IN := FALSE;
		
		FOR byLPForInverter := 1 TO 30 BY 1 DO 
			arrDataSymo10[byLPForInverter].bFunctionIsActive := FALSE;
				arrDataSymo10[byLPForInverter].eOperatingStateInverter := E_Symo_PV_OperatingState.eNoDataReceived;
					arrDataSymo10[byLPForInverter].lrPowerAcInverter := 0;
			arrCurrentL1[byLPForInverter] := 0;
				arrCurrentL2[byLPForInverter] := 0;
			arrCurrentL3[byLPForInverter] := 0;
				arrVoltageL1L2[byLPForInverter] := 0;
			arrVoltageL2L3[byLPForInverter] := 0;
				arrVoltageL3L1[byLPForInverter] := 0;
			arrVoltageL1N[byLPForInverter] := 0;
				arrVoltageL2N[byLPForInverter] := 0;
			arrVoltageL3N[byLPForInverter] := 0;
				arrACPower[byLPForInverter] := 0;
			arrFrequency[byLPForInverter] := 0;
				arrApparentPower[byLPForInverter] := 0;
			arrReactivePower[byLPForInverter] := 0;
				arrProductionEnergy[byLPForInverter] := 0;
		END_FOR
				fbMBRead_FC3.bExecute := FALSE;
					lrCheckValue := 0;
			
		//After reset the Arrays when we have a change on the Unit ID's we restart the State Machine
		IF MEMCMP(ADR(arrUnitID_Inverter),ADR(arrUnitID_Inverter_CP),SIZEOF(arrUnitID_Inverter_CP)) <> 0 AND bEnable AND byTotalInverter > 0 THEN
			iStateModbus := 1;
				arrUnitID_Inverter_CP := arrUnitID_Inverter;
		END_IF
		
	1://Search the Unit ID to read out the Data for each Inverter with Unit ID <> 0
		iStateModbus_CP := iStateModbus;
		
		IF byInverterInProgress >= 30 THEN byInverterInProgress := 0; END_IF
		
		byInverterInProgress := byInverterInProgress + 1;
			byInverterInProgress := LIMIT(1,byInverterInProgress,30);	
		
		IF arrUnitID_Inverter[byInverterInProgress] <> 0 THEN iStateModbus := 2; END_IF
				
	2://Read out first Registers from 40072 to 40118
		arrDataSymo10[byInverterInProgress].bFunctionIsActive := TRUE;
			iStateModbus_CP := iStateModbus;
		
		fbMBRead_FC3.nQuantity := 47;
			fbMBRead_FC3.nMBAddr := 40071;
				fbMBRead_FC3.bExecute := TRUE;
					fbMBRead_FC3.nUnitID := arrUnitID_Inverter[byInverterInProgress];
			
		IF fbMBRead_FC3.bBusy THEN timDelay.IN := TRUE; END_IF
		
		//Wait for Delay, copy Data and then next step
		IF NOT fbMBRead_FC3.bBusy AND NOT fbMBRead_FC3.bError AND timDelay.Q THEN
			//Copy Data Current L1
			fbConvertEnergyRegister(wInputValue_1:= arrBuffer_FC3[3], wInputValue_2:= arrBuffer_FC3[4], eByteOrderForConvert:= eByteOrder.eBigEndian, dwOutputValue=> );
				stFloat.dwRawValue := fbConvertEnergyRegister.dwOutputValue;
					lrCheckValue := stFloat.rValueFloat;	
						IF lrCheckValue >= - 3.402823E+38 AND lrCheckValue <= 3.402823E+38 THEN 
							arrCurrentL1[byInverterInProgress] := lrCheckValue;
						ELSE
							iStateModbus := 300;
								arrDataSymo10[byInverterInProgress].eErrorState := E_Symo_PV_Error.eSymo10TooBigValueReceived;		
						END_IF
			//Copy Data Current L2
			fbConvertEnergyRegister(wInputValue_1:= arrBuffer_FC3[5], wInputValue_2:= arrBuffer_FC3[6], eByteOrderForConvert:= eByteOrder.eBigEndian, dwOutputValue=> );
				stFloat.dwRawValue := fbConvertEnergyRegister.dwOutputValue;
					lrCheckValue := stFloat.rValueFloat;	
						IF lrCheckValue >= - 3.402823E+38 AND lrCheckValue <= 3.402823E+38 THEN 
							arrCurrentL2[byInverterInProgress] := lrCheckValue;
						ELSE
							iStateModbus := 300;
								arrDataSymo10[byInverterInProgress].eErrorState := E_Symo_PV_Error.eSymo10TooBigValueReceived;		
						END_IF
			//Copy Data Current L3
			fbConvertEnergyRegister(wInputValue_1:= arrBuffer_FC3[7], wInputValue_2:= arrBuffer_FC3[8], eByteOrderForConvert:= eByteOrder.eBigEndian, dwOutputValue=> );
				stFloat.dwRawValue := fbConvertEnergyRegister.dwOutputValue;
					lrCheckValue := stFloat.rValueFloat;	
						IF lrCheckValue >= - 3.402823E+38 AND lrCheckValue <= 3.402823E+38 THEN 
							arrCurrentL3[byInverterInProgress] := lrCheckValue;
						ELSE
							iStateModbus := 300;
								arrDataSymo10[byInverterInProgress].eErrorState := E_Symo_PV_Error.eSymo10TooBigValueReceived;		
						END_IF
			//Copy Data Voltage L1-L2
			fbConvertEnergyRegister(wInputValue_1:= arrBuffer_FC3[9], wInputValue_2:= arrBuffer_FC3[10], eByteOrderForConvert:= eByteOrder.eBigEndian, dwOutputValue=> );
				stFloat.dwRawValue := fbConvertEnergyRegister.dwOutputValue;
					lrCheckValue := stFloat.rValueFloat;	
						IF lrCheckValue >= - 3.402823E+38 AND lrCheckValue <= 3.402823E+38 THEN 
							arrVoltageL1L2[byInverterInProgress] := lrCheckValue;
						ELSE
							iStateModbus := 300;
								arrDataSymo10[byInverterInProgress].eErrorState := E_Symo_PV_Error.eSymo10TooBigValueReceived;		
						END_IF
			//Copy Data Voltage L2-L3
			fbConvertEnergyRegister(wInputValue_1:= arrBuffer_FC3[11], wInputValue_2:= arrBuffer_FC3[12], eByteOrderForConvert:= eByteOrder.eBigEndian, dwOutputValue=> );
				stFloat.dwRawValue := fbConvertEnergyRegister.dwOutputValue;
					lrCheckValue := stFloat.rValueFloat;	
						IF lrCheckValue >= - 3.402823E+38 AND lrCheckValue <= 3.402823E+38 THEN 
							arrVoltageL2L3[byInverterInProgress] := lrCheckValue;
						ELSE
							iStateModbus := 300;
								arrDataSymo10[byInverterInProgress].eErrorState := E_Symo_PV_Error.eSymo10TooBigValueReceived;		
						END_IF
			//Copy Data Voltage L3-L1
			fbConvertEnergyRegister(wInputValue_1:= arrBuffer_FC3[13], wInputValue_2:= arrBuffer_FC3[14], eByteOrderForConvert:= eByteOrder.eBigEndian, dwOutputValue=> );
				stFloat.dwRawValue := fbConvertEnergyRegister.dwOutputValue;
					lrCheckValue := stFloat.rValueFloat;	
						IF lrCheckValue >= - 3.402823E+38 AND lrCheckValue <= 3.402823E+38 THEN 
							arrVoltageL3L1[byInverterInProgress] := lrCheckValue;
						ELSE
							iStateModbus := 300;
								arrDataSymo10[byInverterInProgress].eErrorState := E_Symo_PV_Error.eSymo10TooBigValueReceived;		
						END_IF
			//Copy Data Voltage L1-N
			fbConvertEnergyRegister(wInputValue_1:= arrBuffer_FC3[15], wInputValue_2:= arrBuffer_FC3[16], eByteOrderForConvert:= eByteOrder.eBigEndian, dwOutputValue=> );
				stFloat.dwRawValue := fbConvertEnergyRegister.dwOutputValue;
					lrCheckValue := stFloat.rValueFloat;	
						IF lrCheckValue >= - 3.402823E+38 AND lrCheckValue <= 3.402823E+38 THEN 
							arrVoltageL1N[byInverterInProgress] := lrCheckValue;
						ELSE
							iStateModbus := 300;
								arrDataSymo10[byInverterInProgress].eErrorState := E_Symo_PV_Error.eSymo10TooBigValueReceived;		
						END_IF
			//Copy Data Voltage L2-N
			fbConvertEnergyRegister(wInputValue_1:= arrBuffer_FC3[17], wInputValue_2:= arrBuffer_FC3[18], eByteOrderForConvert:= eByteOrder.eBigEndian, dwOutputValue=> );
				stFloat.dwRawValue := fbConvertEnergyRegister.dwOutputValue;
					lrCheckValue := stFloat.rValueFloat;	
						IF lrCheckValue >= - 3.402823E+38 AND lrCheckValue <= 3.402823E+38 THEN 
							arrVoltageL2N[byInverterInProgress] := lrCheckValue;
						ELSE
							iStateModbus := 300;
								arrDataSymo10[byInverterInProgress].eErrorState := E_Symo_PV_Error.eSymo10TooBigValueReceived;		
						END_IF
			//Copy Data Voltage L3-N
			fbConvertEnergyRegister(wInputValue_1:= arrBuffer_FC3[19], wInputValue_2:= arrBuffer_FC3[20], eByteOrderForConvert:= eByteOrder.eBigEndian, dwOutputValue=> );
				stFloat.dwRawValue := fbConvertEnergyRegister.dwOutputValue;
					lrCheckValue := stFloat.rValueFloat;	
						IF lrCheckValue >= - 3.402823E+38 AND lrCheckValue <= 3.402823E+38 THEN 
							arrVoltageL3N[byInverterInProgress] := lrCheckValue;
						ELSE
							iStateModbus := 300;
								arrDataSymo10[byInverterInProgress].eErrorState := E_Symo_PV_Error.eSymo10TooBigValueReceived;		
						END_IF
			//Copy Data AC Power
			fbConvertEnergyRegister(wInputValue_1:= arrBuffer_FC3[21], wInputValue_2:= arrBuffer_FC3[22], eByteOrderForConvert:= eByteOrder.eBigEndian, dwOutputValue=> );
				stFloat.dwRawValue := fbConvertEnergyRegister.dwOutputValue;
					lrCheckValue := stFloat.rValueFloat;	
						IF lrCheckValue >= - 3.402823E+38 AND lrCheckValue <= 3.402823E+38 THEN 
							arrACPower[byInverterInProgress] := lrCheckValue;
								arrDataSymo10[byInverterInProgress].lrPowerAcInverter := arrACPower[byInverterInProgress] / 1000;
						ELSE
							iStateModbus := 300;
								arrDataSymo10[byInverterInProgress].eErrorState := E_Symo_PV_Error.eSymo10TooBigValueReceived;		
						END_IF
			//Copy Data Frequency
			fbConvertEnergyRegister(wInputValue_1:= arrBuffer_FC3[23], wInputValue_2:= arrBuffer_FC3[24], eByteOrderForConvert:= eByteOrder.eBigEndian, dwOutputValue=> );
				stFloat.dwRawValue := fbConvertEnergyRegister.dwOutputValue;
					lrCheckValue := stFloat.rValueFloat;	
						IF lrCheckValue >= - 3.402823E+38 AND lrCheckValue <= 3.402823E+38 THEN 
							arrFrequency[byInverterInProgress] := lrCheckValue;
						ELSE
							iStateModbus := 300;
								arrDataSymo10[byInverterInProgress].eErrorState := E_Symo_PV_Error.eSymo10TooBigValueReceived;		
						END_IF
			//Copy Data Apparent Power
			fbConvertEnergyRegister(wInputValue_1:= arrBuffer_FC3[25], wInputValue_2:= arrBuffer_FC3[26], eByteOrderForConvert:= eByteOrder.eBigEndian, dwOutputValue=> );
				stFloat.dwRawValue := fbConvertEnergyRegister.dwOutputValue;
					lrCheckValue := stFloat.rValueFloat;	
						IF lrCheckValue >= - 3.402823E+38 AND lrCheckValue <= 3.402823E+38 THEN 
							arrApparentPower[byInverterInProgress] := lrCheckValue;
						ELSE
							iStateModbus := 300;
								arrDataSymo10[byInverterInProgress].eErrorState := E_Symo_PV_Error.eSymo10TooBigValueReceived;		
						END_IF
			//Copy Data Reactive Power
			fbConvertEnergyRegister(wInputValue_1:= arrBuffer_FC3[27], wInputValue_2:= arrBuffer_FC3[28], eByteOrderForConvert:= eByteOrder.eBigEndian, dwOutputValue=> );
				stFloat.dwRawValue := fbConvertEnergyRegister.dwOutputValue;
					lrCheckValue := stFloat.rValueFloat;	
						IF lrCheckValue >= - 3.402823E+38 AND lrCheckValue <= 3.402823E+38 THEN 
							arrReactivePower[byInverterInProgress] := lrCheckValue;
						ELSE
							iStateModbus := 300;
								arrDataSymo10[byInverterInProgress].eErrorState := E_Symo_PV_Error.eSymo10TooBigValueReceived;		
						END_IF
			//Copy Data AC production Energy
			fbConvertEnergyRegister(wInputValue_1:= arrBuffer_FC3[31], wInputValue_2:= arrBuffer_FC3[32], eByteOrderForConvert:= eByteOrder.eBigEndian, dwOutputValue=> );
				stFloat.dwRawValue := fbConvertEnergyRegister.dwOutputValue;
					lrCheckValue := stFloat.rValueFloat;	
						IF lrCheckValue >= - 3.402823E+38 AND lrCheckValue <= 3.402823E+38 THEN 
							arrProductionEnergy[byInverterInProgress] := lrCheckValue / 1000;
						ELSE
							iStateModbus := 300;
								arrDataSymo10[byInverterInProgress].eErrorState := E_Symo_PV_Error.eSymo10TooBigValueReceived;		
						END_IF
			//Operating State		
			IF arrBuffer_FC3[47] = 1 THEN arrDataSymo10[byInverterInProgress].eOperatingStateInverter := E_Symo_PV_OperatingState.eOff;
				ELSIF arrBuffer_FC3[47] = 2 THEN arrDataSymo10[byInverterInProgress].eOperatingStateInverter := E_Symo_PV_OperatingState.eSleeping;
				ELSIF arrBuffer_FC3[47] = 3 THEN arrDataSymo10[byInverterInProgress].eOperatingStateInverter := E_Symo_PV_OperatingState.eStartingUp;
				ELSIF arrBuffer_FC3[47] = 4 THEN arrDataSymo10[byInverterInProgress].eOperatingStateInverter := E_Symo_PV_OperatingState.eTrackingPowerPoint;
				ELSIF arrBuffer_FC3[47] = 5 THEN arrDataSymo10[byInverterInProgress].eOperatingStateInverter := E_Symo_PV_OperatingState.eForcedPowerReduction;
				ELSIF arrBuffer_FC3[47] = 6 THEN arrDataSymo10[byInverterInProgress].eOperatingStateInverter := E_Symo_PV_OperatingState.eShuttingDown;
				ELSIF arrBuffer_FC3[47] = 7 THEN arrDataSymo10[byInverterInProgress].eOperatingStateInverter := E_Symo_PV_OperatingState.eFaults;
				ELSIF arrBuffer_FC3[47] = 8 THEN arrDataSymo10[byInverterInProgress].eOperatingStateInverter := E_Symo_PV_OperatingState.eStandby;
				ELSE arrDataSymo10[byInverterInProgress].eOperatingStateInverter := E_Symo_PV_OperatingState.eNoDataReceived;
			END_IF
			//Next Step
			IF iStateModbus = 2 THEN
				fbMBRead_FC3.bExecute := FALSE;
					timDelay.IN := FALSE;
						iStateModbus := 3;
							arrDataSymo10[byInverterInProgress].bError := FALSE; 
								arrDataSymo10[byInverterInProgress].eErrorState := E_Symo_PV_Error.eNoError;
			END_IF
		END_IF
			
		//Error from Inverter
		IF NOT fbMBRead_FC3.bBusy AND NOT fbMBRead_FC3.bError AND timDelay.Q AND arrDataSymo10[byInverterInProgress].eOperatingStateInverter = E_Symo_PV_OperatingState.eFaults THEN
			iStateModbus := 300;
				arrDataSymo10[byInverterInProgress].eErrorState := E_Symo_PV_Error.eSymo10Error;
		END_IF
	 
		//Error or Timeout
		IF FPError_FC_3.Q OR timTimeout.Q THEN
			iStateModbus := 300;
				arrDataSymo10[byInverterInProgress].eErrorState := E_Symo_PV_Error.eModbusTCPError;
		END_IF

	3://Calculate the sum of the values
		iStateModbus_CP := iStateModbus;
		
		lrCounterEnergyProduction := 0;
			fbElMeter.lrCurrentL1 := 0;
		fbElMeter.lrCurrentL2 := 0;	
			fbElMeter.lrCurrentL3 := 0;
		fbElMeter.lrVoltageL1N := 0;
			fbElMeter.lrVoltageL2N := 0;
		fbElMeter.lrVoltageL3N := 0;
			fbElMeter.lrVoltageL1L2 := 0;
		fbElMeter.lrVoltageL2L3 := 0;
			fbElMeter.lrVoltageL3L1 := 0;
		fbElMeter.lrPowerTotal := 0;
			fbElMeter.lrFrequency := 0;
		fbElMeter.lrReactivePowerTotal := 0;
			fbElMeter.lrApparentPowerTotal := 0;
		
		FOR byLPForInverter := 1 TO 30 BY 1 DO 
			lrCounterEnergyProduction := lrCounterEnergyProduction + arrProductionEnergy[byLPForInverter];
			IF lrCounterEnergyProduction > fbElMeter.lrCounterEnergyT1_Production THEN
				fbElMeter.lrCounterEnergyT1_Production := lrCounterEnergyProduction;
			END_IF
				fbElMeter.lrCurrentL1 := fbElMeter.lrCurrentL1 + arrCurrentL1[byLPForInverter];
			fbElMeter.lrCurrentL2 := fbElMeter.lrCurrentL2 + arrCurrentL2[byLPForInverter];	
				fbElMeter.lrCurrentL3 := fbElMeter.lrCurrentL3 + arrCurrentL3[byLPForInverter];
			IF byTotalInverter > 0 THEN
				fbElMeter.lrVoltageL1N := (fbElMeter.lrVoltageL1N + arrVoltageL1N[byLPForInverter]) / byTotalInverter;
					fbElMeter.lrVoltageL2N := (fbElMeter.lrVoltageL2N + arrVoltageL2N[byLPForInverter]) / byTotalInverter;
				fbElMeter.lrVoltageL3N := (fbElMeter.lrVoltageL3N + arrVoltageL3N[byLPForInverter]) / byTotalInverter;
					fbElMeter.lrVoltageL1L2 := (fbElMeter.lrVoltageL1L2 + arrVoltageL1L2[byLPForInverter]) / byTotalInverter;
				fbElMeter.lrVoltageL2L3 := (fbElMeter.lrVoltageL2L3 + arrVoltageL2L3[byLPForInverter]) / byTotalInverter;
					fbElMeter.lrVoltageL3L1 := (fbElMeter.lrVoltageL3L1 + arrVoltageL3L1[byLPForInverter]) / byTotalInverter;
				fbElMeter.lrFrequency := (fbElMeter.lrFrequency + arrFrequency[byLPForInverter]) / byTotalInverter;
			END_IF
					fbElMeter.lrPowerTotal := fbElMeter.lrPowerTotal + arrACPower[byLPForInverter];
				fbElMeter.lrReactivePowerTotal := fbElMeter.lrReactivePowerTotal + arrReactivePower[byLPForInverter];
					fbElMeter.lrApparentPowerTotal := fbElMeter.lrApparentPowerTotal + arrApparentPower[byLPForInverter];
		END_FOR	
					
		fbElMeter.lrTotalCounterEnergy_Production := fbElMeter.lrCounterEnergyT1_Production; 
		
			iStateModbus := 1;
				
	300://Error
		iStateModbus_CP := iStateModbus;
			timDelay.IN := FALSE;
				fbMBRead_FC3.bExecute := FALSE;
					arrDataSymo10[byInverterInProgress].bError := TRUE;
						iStateModbus := 1;				
							
END_CASE

(*------------------------------------------------------------------------------------------Modbus TCP Function---------------------------------------------------------------------------------------------*)

fbMBRead_FC3(sIPAddr:= sIPAdress, nTCPPort:= 502, cbLength:= SIZEOF(arrBuffer_FC3), pDestAddr:= ADR(arrBuffer_FC3), tTimeout:= T#10S );
	FPError_FC_3(CLK:= fbMBRead_FC3.bError, Q=> );

(*----------------------------------------------------------------------------------------Electric Meter Data----------------------------------------------------------------------------------------------*)

//Error and Warning
bErrorDevice := FALSE;
	FOR byLPForInverter := 1 TO 30 BY 1 DO
		IF arrDataSymo10[byLPForInverter].bError THEN bErrorDevice := TRUE; END_IF 
	END_FOR 

IF timDissableFunctions.Q THEN fbElMeter.bWarning := TRUE; fbElMeter.iWarningCode := 0; ELSE fbElMeter.bWarning := FALSE; END_IF   
	IF bErrorDevice OR Lynus_Standards.GVL_Energy.stNumberOfDevices.diNumberOfElectricMeters > Constants_Energy.diMaxNumberOfElectricMeters THEN fbElMeter.bError := TRUE; ELSE fbElMeter.bError := FALSE; END_IF  

IF Lynus_Standards.GVL_Energy.stNumberOfDevices.diNumberOfElectricMeters > Constants_Energy.diMaxNumberOfElectricMeters THEN fbElMeter.iErrorCode := 1;
ELSIF bErrorDevice THEN fbElMeter.iErrorCode := 0;
END_IF  

//Read Out Data done for EM Function
IF iStateModbus <> 3 THEN fbElMeter.bReadOutDataDone := TRUE; ELSE fbElMeter.bReadOutDataDone := FALSE; END_IF

//Function block for meter data
fbElMeter(
	bEnable:= bEnable AND NOT timDissableFunctions.Q, 
	bError:= , 
	bEnableReadOutFunction:= FALSE, 
	bWriteWithDelay:= TRUE,
	bPowerDataInvers:= TRUE, 
	bReadOutDataDone:= ,
	iTimeReadOutInterval:= , 
	iErrorCode:= , 
	iWarningCode:= , 
	lrTotalCounterEnergy_Consumption:= 0, 
	lrTotalCounterEnergy_Production:= , 
	lrCounterEnergyT1_Consumption:= 0, 
	lrCounterEnergyT2_Consumption:= 0, 
	lrCounterEnergyT1_Production:= , 
	lrCounterEnergyT2_Production:= 0, 
	lrCurrentL1:= , 
	lrVoltageL1N:= , 
	lrVoltageL1L2:= , 
	lrPowerL1:= 0, 
	lrCurrentL2:= , 
	lrVoltageL2N:= , 
	lrVoltageL2L3:= , 
	lrPowerL2:= 0, 
	lrCurrentL3:= , 
	lrVoltageL3N:= , 
	lrVoltageL3L1:= , 
	lrPowerL3:= 0, 
	lrPowerTotal:= , 
	lrFrequency:= , 
	lrReactivePowerTotal:= , 
	lrApparentPowerTotal:= , 
	tTimDelayOutput:= T#5S, 
	stDataEMOutPower=> , 
	stDataEMOutPowerDelay=> stDataEMPower_PV, 
	stDataEMOutCounter=> ,
	stDataEMOutCounterDelay=> stDataEMCounter_PV, 
	bReadOutMeter=> );

(*-----------------------------------------------------------Handle data to Global structure for the Electric Meter system-----------------------------------------------------------------*)

CASE iStateGVLData OF
	
	0://Init Step
		byWaitInStep := 0;
			diCounterForGVL := 1;
	
	1://Wait for 4 Steps before clean al Data on GVL
		byWaitInStep := byWaitInStep + 1;
			IF byWaitInStep >= 4 AND fbNumberDevice.bNumberIsCalculatet THEN iStateGVLData := 2; END_IF
				//To much Devices, back to the Init step
				IF byWaitInStep >= 4 AND NOT fbNumberDevice.bNumberIsCalculatet THEN iStateGVLData := 0; END_IF	
			
	2://Clear all Data in GVL
		Lynus_Standards.GVL_Energy.stDataElectricMeters[diCounterForGVL].bEnabled := FALSE;	
			Lynus_Standards.GVL_Energy.stDataElectricMeters[diCounterForGVL].byErrorWarning := 0;
				Lynus_Standards.GVL_Energy.stDataElectricMeters[diCounterForGVL].lrCounterEnergyT1_Consumption := 0;
					Lynus_Standards.GVL_Energy.stDataElectricMeters[diCounterForGVL].lrCounterEnergyT1_Production := 0;
						Lynus_Standards.GVL_Energy.stDataElectricMeters[diCounterForGVL].lrCounterEnergyT2_Consumption := 0;
							Lynus_Standards.GVL_Energy.stDataElectricMeters[diCounterForGVL].lrCounterEnergyT2_Production := 0;
								Lynus_Standards.GVL_Energy.stDataElectricMeters[diCounterForGVL].lrPower := 0;
									Lynus_Standards.GVL_Energy.stDataElectricMeters[diCounterForGVL].lrPowerConsumption := 0;
										Lynus_Standards.GVL_Energy.stDataElectricMeters[diCounterForGVL].lrPowerConsumption := 0;
											Lynus_Standards.GVL_Energy.stDataElectricMeters[diCounterForGVL].lrPowerProduction := 0;
												Lynus_Standards.GVL_Energy.stDataElectricMeters[diCounterForGVL].lrTotalCounterEnergy_Consumption := 0;
													Lynus_Standards.GVL_Energy.stDataElectricMeters[diCounterForGVL].lrTotalCounterEnergy_Production := 0;
		
		diCounterForGVL := diCounterForGVL + 1;
			diCounterForGVL := LIMIT(0,diCounterForGVL,Constants_Energy.diMaxNumberOfElectricMeters);
				//Back to the init step
				IF diCounterForGVL >= Constants_Energy.diMaxNumberOfElectricMeters THEN iStateGVLData := 0; END_IF

END_CASE 	 

IF diNrOfEM_OUT_PV > 0 AND fbNumberDevice.bNumberIsCalculatet THEN
	Lynus_Standards.GVL_Energy.stDataElectricMeters[diNrOfEM_OUT_PV].bEnabled := fbElMeter.stDataEMOutPower.bEnabled;
		Lynus_Standards.GVL_Energy.stDataElectricMeters[diNrOfEM_OUT_PV].byErrorWarning := fbElMeter.stDataEMOutPower.byErrorWarning;
			Lynus_Standards.GVL_Energy.stDataElectricMeters[diNrOfEM_OUT_PV].lrCounterEnergyT1_Consumption := fbElMeter.stDataEMOutCounter.lrCounterEnergyT1_Consumption;
				Lynus_Standards.GVL_Energy.stDataElectricMeters[diNrOfEM_OUT_PV].lrCounterEnergyT1_Production := fbElMeter.stDataEMOutCounter.lrCounterEnergyT1_Production;
					Lynus_Standards.GVL_Energy.stDataElectricMeters[diNrOfEM_OUT_PV].lrCounterEnergyT2_Consumption := fbElMeter.stDataEMOutCounter.lrCounterEnergyT2_Consumption;
						Lynus_Standards.GVL_Energy.stDataElectricMeters[diNrOfEM_OUT_PV].lrCounterEnergyT2_Production := fbElMeter.stDataEMOutCounter.lrCounterEnergyT2_Production;		
							Lynus_Standards.GVL_Energy.stDataElectricMeters[diNrOfEM_OUT_PV].lrPower := fbElMeter.stDataEMOutPower.lrPowerTotal;
								Lynus_Standards.GVL_Energy.stDataElectricMeters[diNrOfEM_OUT_PV].lrPowerConsumption := fbElMeter.stDataEMOutPower.lrPowerConsumption;
									Lynus_Standards.GVL_Energy.stDataElectricMeters[diNrOfEM_OUT_PV].lrPowerProduction := fbElMeter.stDataEMOutPower.lrPowerProduction;
										Lynus_Standards.GVL_Energy.stDataElectricMeters[diNrOfEM_OUT_PV].lrTotalCounterEnergy_Consumption := fbElMeter.stDataEMOutCounter.lrTotalCounterEnergy_Consumption;
											Lynus_Standards.GVL_Energy.stDataElectricMeters[diNrOfEM_OUT_PV].lrTotalCounterEnergy_Production := fbElMeter.stDataEMOutCounter.lrTotalCounterEnergy_Production;
END_IF

(*----------------------------------------------------------Save persistent data----------------------------------------------------------------*)

arrPD[1](lrValue:= BOOL_TO_LREAL(bEnable), bEventBasedActive=> );
arrPD[2](lrValue:= BYTE_TO_LREAL(arrUnitID_Inverter[1]), bEventBasedActive=> );
arrPD[3](lrValue:= BYTE_TO_LREAL(arrUnitID_Inverter[2]), bEventBasedActive=> );
arrPD[4](lrValue:= BYTE_TO_LREAL(arrUnitID_Inverter[3]), bEventBasedActive=> );
arrPD[5](lrValue:= BYTE_TO_LREAL(arrUnitID_Inverter[4]), bEventBasedActive=> );
arrPD[6](lrValue:= BYTE_TO_LREAL(arrUnitID_Inverter[5]), bEventBasedActive=> );
arrPD[7](lrValue:= BYTE_TO_LREAL(arrUnitID_Inverter[6]), bEventBasedActive=> );
arrPD[8](lrValue:= BYTE_TO_LREAL(arrUnitID_Inverter[7]), bEventBasedActive=> );
arrPD[9](lrValue:= BYTE_TO_LREAL(arrUnitID_Inverter[8]), bEventBasedActive=> );
arrPD[10](lrValue:= BYTE_TO_LREAL(arrUnitID_Inverter[9]), bEventBasedActive=> );
arrPD[11](lrValue:= BYTE_TO_LREAL(arrUnitID_Inverter[10]), bEventBasedActive=> );
arrPD[12](lrValue:= BYTE_TO_LREAL(arrUnitID_Inverter[11]), bEventBasedActive=> );
arrPD[13](lrValue:= BYTE_TO_LREAL(arrUnitID_Inverter[12]), bEventBasedActive=> );
arrPD[14](lrValue:= BYTE_TO_LREAL(arrUnitID_Inverter[13]), bEventBasedActive=> );
arrPD[15](lrValue:= BYTE_TO_LREAL(arrUnitID_Inverter[14]), bEventBasedActive=> );
arrPD[16](lrValue:= BYTE_TO_LREAL(arrUnitID_Inverter[15]), bEventBasedActive=> );
arrPD[17](lrValue:= BYTE_TO_LREAL(arrUnitID_Inverter[16]), bEventBasedActive=> );
arrPD[18](lrValue:= BYTE_TO_LREAL(arrUnitID_Inverter[17]), bEventBasedActive=> );
arrPD[19](lrValue:= BYTE_TO_LREAL(arrUnitID_Inverter[18]), bEventBasedActive=> );
arrPD[20](lrValue:= BYTE_TO_LREAL(arrUnitID_Inverter[19]), bEventBasedActive=> );
arrPD[21](lrValue:= BYTE_TO_LREAL(arrUnitID_Inverter[20]), bEventBasedActive=> );
arrPD[22](lrValue:= BYTE_TO_LREAL(arrUnitID_Inverter[21]), bEventBasedActive=> );
arrPD[23](lrValue:= BYTE_TO_LREAL(arrUnitID_Inverter[22]), bEventBasedActive=> );
arrPD[24](lrValue:= BYTE_TO_LREAL(arrUnitID_Inverter[23]), bEventBasedActive=> );
arrPD[25](lrValue:= BYTE_TO_LREAL(arrUnitID_Inverter[24]), bEventBasedActive=> );
arrPD[26](lrValue:= BYTE_TO_LREAL(arrUnitID_Inverter[25]), bEventBasedActive=> );
arrPD[27](lrValue:= BYTE_TO_LREAL(arrUnitID_Inverter[26]), bEventBasedActive=> );
arrPD[28](lrValue:= BYTE_TO_LREAL(arrUnitID_Inverter[27]), bEventBasedActive=> );
arrPD[29](lrValue:= BYTE_TO_LREAL(arrUnitID_Inverter[28]), bEventBasedActive=> );
arrPD[30](lrValue:= BYTE_TO_LREAL(arrUnitID_Inverter[29]), bEventBasedActive=> );
arrPD[31](lrValue:= BYTE_TO_LREAL(arrUnitID_Inverter[30]), bEventBasedActive=> );
PD_String(sText:= sIPAdress, bEventBasedActive=> );

END_FUNCTION_BLOCK
